PROGRAM MAIN
VAR
	
MyController : Controller;  

			
END_VAR

MyController.Motion_Parameters.maxVelocity := 800;

MyController.NumberOfXTiles := 4;
MyController.NumberOfYTiles := 3;
MyController.MoverType := 4330;
MyController.HapticfeedBack := TRUE; 

MyController();

END_PROGRAM

(* stored: Version 1.1.0.1, ProductVersion 3.1.4024.12
   POU MAIN: Id {fe375bac-6b9b-4870-b48c-47a23cbcf2e8}, SpecialFunc None *)
